(* PLC project BitString_Operators.project, CODESYS CODESYS V3.5 SP18 Patch 3 *)
(* stored: creationDateTime 2025-01-01T18:30:19.1932179, modificationDateTime 2025-01-01T18:29:48.5883786 *)

FUNCTION_BLOCK FB_OrElse
  VAR
    iCounter : INT;
  END_VAR

            
          

METHOD TestMethod : BOOL
                  iCounter := iCounter + 1;
TestMethod := TRUE;
                
END_METHOD
END_FUNCTION_BLOCK

PROGRAM Bitstring_Operators
  VAR
    fbSampleOrElse : FB_OrElse;  (* Or_Else *)
    xResult : BOOL;
    xVar : BOOL;
    pxSensor : POINTER TO BOOL;  (* Pointer to a sensor (can be NULL if not initialized) *)
    xAlarm : BOOL;  (* Variable to activate the alarm *)
    wVarAnd : WORD;  (* And *)
    wVarOr : WORD;  (* Or *)
    wVarXor : WORD;  (* Xor *)
    wVarNot : WORD;  (* Not *)
  END_VAR

            _And();
_And_Then();
_Or();
_Or_Else();
_Not();
_Xor();

          

ACTION _Or_Else:
                xResult := xVar OR_ELSE fbSampleOrElse.TestMethod();
//Counter of fbSampleOrElse does not increases as the method is not executed
              
END_ACTION

ACTION _And:
                wVarAnd := 2#1001_0011 AND 2#1000_1010;
	(* Result in wVarAnd: 2#1000_0010 *)
              
END_ACTION

ACTION _Or:
                wVarOr:= 2#1001_0011 OR 2#1000_1010;
	(* Result in wVarOr: 2#1001_1011 *)
              
END_ACTION

ACTION _Not:
                wVarNot := NOT 2#1001_0011;
	(* Result in wVarNot: 2#0110_1100 *)
              
END_ACTION

ACTION _And_Then:
                (*	pxSensor := ADR(xSomethingSensor);     pSensor points to xSomethingSensor *)
IF (pxSensor <> 0 AND_THEN pxSensor^) THEN 
    (* Additional logic can be implemented below *)
    xAlarm := TRUE;
END_IF

(*  
	If we used AND instead of AND_THEN, the program would 
    attempt to access pSensor^ even if pSensor is 0, which 
    would cause a runtime error. Therefore, using AND_THEN 
    is safer and more efficient in this case.
*)

              
END_ACTION

ACTION _Xor:
                wVarXor := 2#1001_0011 XOR 2#1000_1010;
		(* Result in wVarXor: 2#1001_0011 *)

              
END_ACTION
END_PROGRAM
